(* IEC 61131-3 sources: horner-cscape-mcp/artifacts/projects/TankLevelFailureTest/pous, 2 files *)

(* ---- TankLevelFailureTest.st ---- *)
PROGRAM TankLevelFailureTest
VAR
    TankLevel : REAL := 50.0;
    TargetLevel : REAL := 60.0;
END_VAR
TargetLevel := TankLevel + ;
END_PROGRAM

(* ---- TankLevelValid.st ---- *)
PROGRAM TankLevelValid
VAR
    TankLevel : REAL := 50.0;
    TargetLevel : REAL := 60.0;
    PumpRun : BOOL := FALSE;
END_VAR

IF TankLevel < TargetLevel THEN
    PumpRun := TRUE;
ELSE
    PumpRun := FALSE;
END_IF;
END_PROGRAM
